PROGRAM MAIN
VAR
	{attribute 'pytmc' := '
        pv: FAT:TEST:BSD
    '}
	M1 : DUT_MotionStage := (nEnableMode:=ENUM_StageEnableMode.ALWAYS, bPowerSelf:=TRUE);
    fbMotionStageM1 : FB_MotionStage;
END_VAR

fbMotionStageM1(stMotionStage:=M1);
m1.bHardwareEnable := True;
m1.bLimitBackwardEnable := True;
m1.bLimitForwardEnable := True;

END_PROGRAM

(* stored: Version 1.1.0.1, ProductVersion 3.1.4024.15
   POU MAIN: Id {be7aa4c0-9182-4858-a218-fa58c2e5f257}, SpecialFunc None *)
